VAR_INPUT
	m_Input_NumTextList:		INT;
END_VAR
    Rectangle (0,0 446x169), "%s", text list: 'TextList_Gaz', text index: m_Input_NumTextList
    Rectangle (361,0 85x25), "%s", text variable: m_Input_DG.CONF_Util_Name
    Frame (3,35 153x52)
        shows VISU_FCTS_SA(m_Input_ID_XML := 12, m_Input_UserRight := PRG_USER.ACTU_USER.FONCTION_SA AND NOT m_Input_Machine.STATE_Prod, m_Input_Operation := m_Input_Ligne.OP_MARCHE)
    Frame (3,106 153x52)
        shows VISU_FCTS_SA(m_Input_ID_XML := 13, m_Input_UserRight := PRG_USER.ACTU_USER.FONCTION_SA AND NOT m_Input_Machine.STATE_Prod, m_Input_Operation := m_Input_Ligne.OP_ARRET)
    Rectangle (170,99 91x24), "%s", text list: 'TextList_Gaz', text index: 3
    RoundedRectangle (354,99 87x24), "%1.1f", text variable: m_Input_DG.STATE_Flow
    RoundedRectangle (263,99 87x24), "%1.1f", text variable: m_Input_Ligne.PRM_Flow, input disabled if: (NOT PRG_USER.ACTU_USER.FONCTION_SA AND NOT m_Input_Machine.STATE_Prod) OR (NOT PRG_USER.ACTU_USER.MODIF_ENLIGNE AND m_Input_Machine.STATE_Prod)
        OnMouseClick: write the text variable via InputWithLimits, min 0, max m_Input_DG.CONF_Util_Max_Flow
    Rectangle (170,132 91x24), "%s", text list: 'TextList_Basiques', text index: 22
    RoundedRectangle (263,132 87x24), "%s", text variable: m_Input_Ligne.OP_RAMPE.PRM_Temps, input disabled if: (NOT PRG_USER.ACTU_USER.FONCTION_SA AND NOT m_Input_Machine.STATE_Prod) OR (NOT PRG_USER.ACTU_USER.MODIF_ENLIGNE AND m_Input_Machine.STATE_Prod)
        OnMouseClick: write the text variable via InputWithLimits
    Frame (163,35 153x52)
        shows VISU_FCTS_SA(m_Input_ID_XML := 14, m_Input_UserRight := PRG_USER.ACTU_USER.FONCTION_SA AND NOT m_Input_Machine.STATE_Prod, m_Input_Operation := m_Input_Ligne.OP_RAMPE.MARCHE)
    Button (323,35 120x50), "%s", input disabled if: (NOT PRG_USER.ACTU_USER.FONCTION_SA AND NOT m_Input_Machine.STATE_Prod) OR (NOT PRG_USER.ACTU_USER.MODIF_ENLIGNE AND m_Input_Machine.STATE_Prod), text list: 'TextList_Basiques', text index: 19
        toggle m_Input_Ligne.CO_Modif
    RoundedRectangle (354,132 87x24), "%s", text variable: m_Input_Ligne.OP_RAMPE.OUT_Tps_ecoule
END_VISUALIZATION

// ---- Visualizations/Semi Auto/Elements/SA_LIGNE_GAZ_MKS_RAMPE.TcVIS
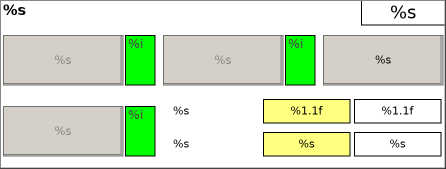
VISUALIZATION SA_LIGNE_GAZ_MKS_RAMPE  // 446x169
VAR_IN_OUT
	m_Input_Ligne:		BLOCK_LIGNE_GAZ;
	m_Input_Machine:	BLOCK_MODE_MARCHE_V2_0;
	m_Input_DG:			BLOCK_MFC_MKS_NoCoE;
	m_Input_UserRight:	BOOL;
END_VAR

VAR_INPUT
	m_Input_NumTextList:		INT;
END_VAR
    Rectangle (0,0 446x169), "%s", text list: 'TextList_Gaz', text index: m_Input_NumTextList
    Rectangle (361,0 85x25), "%s", text variable: m_Input_DG.CONF_Util_Name
    Frame (3,35 153x52)
        shows VISU_FCTS_SA(m_Input_ID_XML := 12, m_Input_UserRight := PRG_USER.ACTU_USER.FONCTION_SA AND NOT m_Input_Machine.STATE_Prod, m_Input_Operation := m_Input_Ligne.OP_MARCHE)
    Frame (3,106 153x52)
        shows VISU_FCTS_SA(m_Input_ID_XML := 13, m_Input_UserRight := PRG_USER.ACTU_USER.FONCTION_SA AND NOT m_Input_Machine.STATE_Prod, m_Input_Operation := m_Input_Ligne.OP_ARRET)
    Rectangle (170,99 91x24), "%s", text list: 'TextList_Gaz', text index: 3
    RoundedRectangle (354,99 87x24), "%1.1f", text variable: m_Input_DG.STATE_Flow
    RoundedRectangle (263,99 87x24), "%1.1f", text variable: m_Input_Ligne.PRM_Flow, input disabled if: (NOT PRG_USER.ACTU_USER.FONCTION_SA AND NOT m_Input_Machine.STATE_Prod) OR (NOT PRG_USER.ACTU_USER.MODIF_ENLIGNE AND m_Input_Machine.STATE_Prod)
        OnMouseClick: write the text variable via InputWithLimits, min 0, max m_Input_DG.CONF_Util_Max_Flow
    Rectangle (170,132 91x24), "%s", text list: 'TextList_Basiques', text index: 22
    RoundedRectangle (263,132 87x24), "%s", text variable: m_Input_Ligne.OP_RAMPE.PRM_Temps, input disabled if: (NOT PRG_USER.ACTU_USER.FONCTION_SA AND NOT m_Input_Machine.STATE_Prod) OR (NOT PRG_USER.ACTU_USER.MODIF_ENLIGNE AND m_Input_Machine.STATE_Prod)
        OnMouseClick: write the text variable via Edit
    Frame (163,35 153x52)
        shows VISU_FCTS_SA(m_Input_ID_XML := 14, m_Input_UserRight := PRG_USER.ACTU_USER.FONCTION_SA AND NOT m_Input_Machine.STATE_Prod, m_Input_Operation := m_Input_Ligne.OP_RAMPE.MARCHE)
    Button (323,35 120x50), "%s", input disabled if: (NOT PRG_USER.ACTU_USER.FONCTION_SA AND NOT m_Input_Machine.STATE_Prod) OR (NOT PRG_USER.ACTU_USER.MODIF_ENLIGNE AND m_Input_Machine.STATE_Prod), text list: 'TextList_Basiques', text index: 19
        toggle m_Input_Ligne.CO_Modif
    RoundedRectangle (354,132 87x24), "%s", text variable: m_Input_Ligne.OP_RAMPE.OUT_Tps_ecoule
END_VISUALIZATION

// ---- Visualizations/Semi Auto/Elements/SA_POMP_1E_PCR_PPM.TcVIS
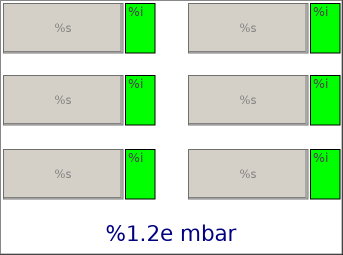
VISUALIZATION SA_POMP_1E_PCR_PPM  // 343x255
VAR_IN_OUT
	m_Input_PRG:		BLOCK_PRG_POMPAGE;
	m_Input_Jauge:		BLOCK_BCG450_ANA;
END_VAR
    Rectangle (0,0 343x255)
    Frame (3,75 153x52)
        shows VISU_FCTS_SA(m_Input_ID_XML := 0, m_Input_UserRight := PRG_USER.ACTU_USER.FONCTION_SA, m_Input_Operation := m_Input_PRG.POMPAGE.OP_Pompage_Sec)
    Frame (3,3 153x52)
        shows VISU_FCTS_SA(m_Input_ID_XML := 1, m_Input_UserRight := PRG_USER.ACTU_USER.FONCTION_SA, m_Input_Operation := m_Input_PRG.POMPAGE.OP_Marche_Pompes)
    Frame (188,3 153x52)
        shows VISU_FCTS_SA(m_Input_ID_XML := 2, m_Input_UserRight := PRG_USER.ACTU_USER.FONCTION_SA, m_Input_Operation := m_Input_PRG.POMPAGE.OP_Arret_Pompes)
    Frame (188,75 153x52)
        shows VISU_FCTS_SA(m_Input_ID_XML := 3, m_Input_UserRight := PRG_USER.ACTU_USER.FONCTION_SA, m_Input_Operation := m_Input_PRG.POMPAGE.OP_Isolement)
    Frame (3,149 153x52)
        shows VISU_FCTS_SA(m_Input_ID_XML := 4, m_Input_UserRight := PRG_USER.ACTU_USER.FONCTION_SA, m_Input_Operation := m_Input_PRG.POMPAGE.OP_Ventilation)
    Rectangle (80,219 182x29), "%1.2e mbar", text variable: m_Input_Jauge.STATE_Pression
    Frame (188,149 153x52)
        shows VISU_FCTS_SA(m_Input_ID_XML := 17, m_Input_UserRight := PRG_USER.ACTU_USER.FONCTION_SA, m_Input_Operation := m_Input_PRG.POMPAGE.OP_Regen)
END_VISUALIZATION

// ---- Visualizations/Semi Auto/Elements/SA_POMP_1E_PCR_PPM_ASS.TcVIS
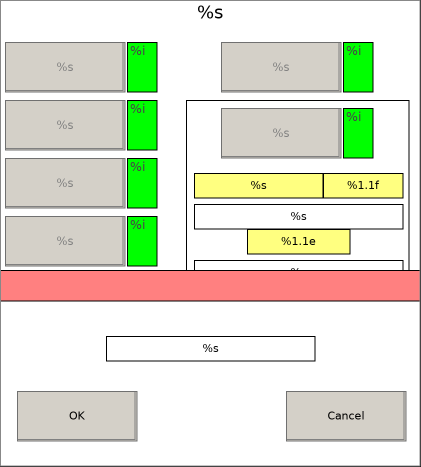
VISUALIZATION SA_POMP_1E_PCR_PPM_ASS  // 421x467
VAR_IN_OUT
	m_Input_PRG:			BLOCK_PRG_POMPAGE;
	m_Input_Jauge:			BLOCK_BCG450_ETHERCAT;
	m_Input_Process:		BLOCK_CDG_ETHERCAT;
	m_Input_Vanne:			BLOCK_VVAT_650_ETHERCAT;
	m_Input_Machine:		BLOCK_MODE_MARCHE_V2_0;
END_VAR
    Rectangle (0,0 421x467), "%s", text list: 'TextList_Navigation', text index: 6
    Frame (5,42 153x52)
        shows VISU_FCTS_SA(m_Input_ID_XML := 1, m_Input_UserRight := PRG_USER.ACTU_USER.FONCTION_SA, m_Input_Operation := m_Input_PRG.POMPAGE.OP_Marche_Pompes)
    Rectangle (74,391 63x25), "%s", text variable: m_Input_Jauge.MNEMO
    Rectangle (144,389 192x29), "%1.2e mbar", text variable: m_Input_Jauge.STATE_Pression
    Rectangle (74,425 63x25), "%s", text variable: m_Input_Process.MNEMO
    Rectangle (144,423 192x29), "%1.2e mbar", text variable: m_Input_Process.STATE_Pression
    Frame (5,100 153x52)
        shows VISU_FCTS_SA(m_Input_ID_XML := 0, m_Input_UserRight := PRG_USER.ACTU_USER.FONCTION_SA, m_Input_Operation := m_Input_PRG.POMPAGE.OP_Pompage_Sec)
    Frame (5,216 153x52)
        shows VISU_FCTS_SA(m_Input_ID_XML := 3, m_Input_UserRight := PRG_USER.ACTU_USER.FONCTION_SA, m_Input_Operation := m_Input_PRG.POMPAGE.OP_Isolement)
    Frame (4,334 153x52)
        shows VISU_FCTS_SA(m_Input_ID_XML := 17, m_Input_UserRight := FALSE, m_Input_Operation := m_Input_PRG.POMPAGE.OP_Regen)
    Frame (5,274 153x52)
        shows VISU_FCTS_SA(m_Input_ID_XML := 4, m_Input_UserRight := PRG_USER.ACTU_USER.FONCTION_SA, m_Input_Operation := m_Input_PRG.POMPAGE.OP_Ventilation)
    Rectangle (186,100 223x274)
    Frame (221,108 153x52)
        shows VISU_FCTS_SA(m_Input_ID_XML := 11, m_Input_UserRight := PRG_USER.ACTU_USER.FONCTION_SA, m_Input_Operation := m_Input_PRG.POMPAGE.OP_Pompage_Proc)
    RoundedRectangle (194,173 129x25), "%s", invisible if: NOT m_Input_Vanne.PRM_Mode, input disabled if: NOT (PRG_USER.ACTU_USER.FONCTION_SA AND NOT m_Input_MACHINE.STATE_Prod) OR m_Input_MACHINE.STATE_Prod, text list: 'TextList_VVAT_650_ETHERCAT', text index: 8
        OnMouseClick: toggle m_Input_Vanne.PRM_Mode
    RoundedRectangle (194,173 129x25), "%s", invisible if: m_Input_Vanne.PRM_Mode, input disabled if: NOT (PRG_USER.ACTU_USER.FONCTION_SA AND NOT m_Input_MACHINE.STATE_Prod) OR m_Input_MACHINE.STATE_Prod, text list: 'TextList_VVAT_650_ETHERCAT', text index: 7
        OnMouseClick: toggle m_Input_Vanne.PRM_Mode
    RoundedRectangle (194,204 209x25), "%s", invisible if: NOT m_Input_Vanne.PRM_Mode, text list: 'TextList_VVAT_650_ETHERCAT', text index: 4
    RoundedRectangle (194,260 209x25), "%s", invisible if: NOT m_Input_Vanne.PRM_Mode, text list: 'TextList_VVAT_650_ETHERCAT', text index: 5
    RoundedRectangle (194,316 209x25), "%s", invisible if: NOT m_Input_Vanne.PRM_Mode, text list: 'TextList_VVAT_650_ETHERCAT', text index: 6
    RoundedRectangle (247,341 103x25), "%s", text variable: m_Input_Vanne.PRM_Tim_W_Pr, invisible if: NOT m_Input_Vanne.PRM_Mode, input disabled if: NOT (PRG_USER.ACTU_USER.FONCTION_SA AND NOT m_Input_MACHINE.STATE_Prod) OR m_Input_MACHINE.STATE_Prod
        OnMouseClick: write the text variable via InputWithLimits
    RoundedRectangle (247,285 103x25), "%1.1e", text variable: m_Input_Vanne.PRM_W_Pr_HI, invisible if: NOT m_Input_Vanne.PRM_Mode, input disabled if: NOT (PRG_USER.ACTU_USER.FONCTION_SA AND NOT m_Input_MACHINE.STATE_Prod) OR m_Input_MACHINE.STATE_Prod
        OnMouseClick: write the text variable via InputWithLimits, min 0, max 1000
    RoundedRectangle (247,229 103x25), "%1.1e", text variable: m_Input_Vanne.PRM_W_Pr_LO, invisible if: NOT m_Input_Vanne.PRM_Mode, input disabled if: NOT (PRG_USER.ACTU_USER.FONCTION_SA AND NOT m_Input_MACHINE.STATE_Prod) OR m_Input_MACHINE.STATE_Prod
        OnMouseClick: write the text variable via InputWithLimits, min 0, max 1000
    RoundedRectangle (323,173 80x25), "%1.1e", text variable: m_Input_Vanne.PRM_Pression, invisible if: NOT m_Input_Vanne.PRM_Mode, input disabled if: NOT (PRG_USER.ACTU_USER.FONCTION_SA AND NOT m_Input_MACHINE.STATE_Prod) OR m_Input_MACHINE.STATE_Prod
        OnMouseClick: write the text variable via InputWithLimits, min 0, max 1000
    RoundedRectangle (323,173 80x25), "%1.1f", text variable: m_Input_Vanne.PRM_Position, invisible if: m_Input_Vanne.PRM_Mode, input disabled if: NOT (PRG_USER.ACTU_USER.FONCTION_SA AND NOT m_Input_MACHINE.STATE_Prod) OR m_Input_MACHINE.STATE_Prod
        OnMouseClick: write the text variable via InputWithLimits, min 0, max 100
    Frame (221,42 153x52)
        shows VISU_FCTS_SA(m_Input_ID_XML := 2, m_Input_UserRight := PRG_USER.ACTU_USER.FONCTION_SA, m_Input_Operation := m_Input_PRG.POMPAGE.OP_Arret_Pompes)
    Frame (5,158 153x52)
        shows VISU_FCTS_SA(m_Input_ID_XML := 28, m_Input_UserRight := PRG_USER.ACTU_USER.FONCTION_SA, m_Input_Operation := m_Input_PRG.POMPAGE.OP_Pompage_Prim)
    Button (4,334 120x50), "%s", input disabled if: NOT m_Input_PRG.POMPAGE.OP_Regen.Autor_IHM OR NOT (PRG_USER.ACTU_USER.FONCTION_SA AND NOT m_Input_Machine.STATE_PROD), text list: 'TextList_SA_Operations', text index: 17
        OnMouseClick: execute { Global_Variables.SHOW_CONFIRM_REGEN:=(TRUE); }
    Group (0,270 421x197), invisible if: NOT Global_Variables.SHOW_CONFIRM_REGEN
        Rectangle (0,0 421x197)
        Button (17,121 120x50), "OK", input disabled if: NOT m_Input_PRG.POMPAGE.OP_Regen.Autor_IHM OR NOT (PRG_USER.ACTU_USER.FONCTION_SA AND NOT m_Input_Machine.STATE_PROD)
            OnMouseClick: execute { m_Input_PRG.POMPAGE.OP_Regen.ON_IHM:=(TRUE); Global_Variables.SHOW_CONFIRM_REGEN:=(FALSE); }
        Button (286,121 120x50), "Cancel"
            OnMouseClick: execute { Global_Variables.SHOW_CONFIRM_REGEN:=(FALSE); }
        Rectangle (0,0 421x31)
        RoundedRectangle (106,66 209x25), "%s", text list: 'TextList_Pompage', text index: 1
END_VISUALIZATION

// ---- Visualizations/Semi Auto/Elements/SA_POMP_1E_PCR_PPM_ASS_M11.TcVIS
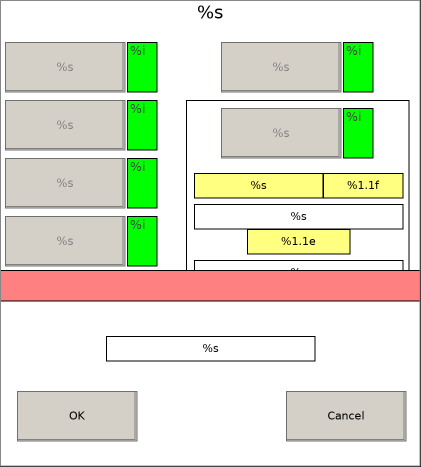
VISUALIZATION SA_POMP_1E_PCR_PPM_ASS_M11  // 421x467
VAR_IN_OUT
	m_Input_PRG:			BLOCK_PRG_POMPAGE;
	m_Input_Jauge:			BLOCK_BCG450_ETHERCAT;
	m_Input_Vanne:			BLOCK_VVAT_650_NO;
	m_Input_Machine:		BLOCK_MODE_MARCHE_V2_0;
END_VAR
    Rectangle (0,0 421x467), "%s", text list: 'TextList_Navigation', text index: 6
    Frame (5,42 153x52)
        shows VISU_FCTS_SA(m_Input_ID_XML := 1, m_Input_UserRight := PRG_USER.ACTU_USER.FONCTION_SA, m_Input_Operation := m_Input_PRG.POMPAGE.OP_Marche_Pompes)
    Rectangle (74,391 63x25), "%s", text variable: m_Input_Jauge.MNEMO
    Rectangle (144,389 192x29), "%1.2e mbar", text variable: m_Input_Jauge.STATE_Pression
    Frame (5,100 153x52)
        shows VISU_FCTS_SA(m_Input_ID_XML := 0, m_Input_UserRight := PRG_USER.ACTU_USER.FONCTION_SA, m_Input_Operation := m_Input_PRG.POMPAGE.OP_Pompage_Sec)
    Frame (5,216 153x52)
        shows VISU_FCTS_SA(m_Input_ID_XML := 3, m_Input_UserRight := PRG_USER.ACTU_USER.FONCTION_SA, m_Input_Operation := m_Input_PRG.POMPAGE.OP_Isolement)
    Frame (4,334 153x52)
        shows VISU_FCTS_SA(m_Input_ID_XML := 17, m_Input_UserRight := FALSE, m_Input_Operation := m_Input_PRG.POMPAGE.OP_Regen)
    Frame (5,274 153x52)
        shows VISU_FCTS_SA(m_Input_ID_XML := 4, m_Input_UserRight := PRG_USER.ACTU_USER.FONCTION_SA, m_Input_Operation := m_Input_PRG.POMPAGE.OP_Ventilation)
    Rectangle (186,100 223x274)
    Frame (221,108 153x52)
        shows VISU_FCTS_SA(m_Input_ID_XML := 11, m_Input_UserRight := PRG_USER.ACTU_USER.FONCTION_SA, m_Input_Operation := m_Input_PRG.POMPAGE.OP_Pompage_Proc)
    RoundedRectangle (194,173 129x25), "%s", invisible if: NOT m_Input_Vanne.PRM_Mode, input disabled if: NOT (PRG_USER.ACTU_USER.FONCTION_SA AND NOT m_Input_MACHINE.STATE_Prod) OR m_Input_MACHINE.STATE_Prod, text list: 'TextList_VVAT_650_ETHERCAT', text index: 8
        OnMouseClick: toggle m_Input_Vanne.PRM_Mode
    RoundedRectangle (194,173 129x25), "%s", invisible if: m_Input_Vanne.PRM_Mode, input disabled if: NOT (PRG_USER.ACTU_USER.FONCTION_SA AND NOT m_Input_MACHINE.STATE_Prod) OR m_Input_MACHINE.STATE_Prod, text list: 'TextList_VVAT_650_ETHERCAT', text index: 7
        OnMouseClick: toggle m_Input_Vanne.PRM_Mode
    RoundedRectangle (194,204 209x25), "%s", invisible if: NOT m_Input_Vanne.PRM_Mode, text list: 'TextList_VVAT_650_ETHERCAT', text index: 4
    RoundedRectangle (194,260 209x25), "%s", invisible if: NOT m_Input_Vanne.PRM_Mode, text list: 'TextList_VVAT_650_ETHERCAT', text index: 5
    RoundedRectangle (194,316 209x25), "%s", invisible if: NOT m_Input_Vanne.PRM_Mode, text list: 'TextList_VVAT_650_ETHERCAT', text index: 6
    RoundedRectangle (247,341 103x25), "%s", text variable: m_Input_Vanne.PRM_Tim_W_Pr, invisible if: NOT m_Input_Vanne.PRM_Mode, input disabled if: NOT (PRG_USER.ACTU_USER.FONCTION_SA AND NOT m_Input_MACHINE.STATE_Prod) OR m_Input_MACHINE.STATE_Prod
        OnMouseClick: write the text variable via InputWithLimits
    RoundedRectangle (247,285 103x25), "%1.1e", text variable: m_Input_Vanne.PRM_W_Pr_HI, invisible if: NOT m_Input_Vanne.PRM_Mode, input disabled if: NOT (PRG_USER.ACTU_USER.FONCTION_SA AND NOT m_Input_MACHINE.STATE_Prod) OR m_Input_MACHINE.STATE_Prod
        OnMouseClick: write the text variable via InputWithLimits, min 0, max 1000
    RoundedRectangle (247,229 103x25), "%1.1e", text variable: m_Input_Vanne.PRM_W_Pr_LO, invisible if: NOT m_Input_Vanne.PRM_Mode, input disabled if: NOT (PRG_USER.ACTU_USER.FONCTION_SA AND NOT m_Input_MACHINE.STATE_Prod) OR m_Input_MACHINE.STATE_Prod
        OnMouseClick: write the text variable via InputWithLimits, min 0, max 1000
    RoundedRectangle (323,173 80x25), "%1.1e", text variable: m_Input_Vanne.PRM_Pression, invisible if: NOT m_Input_Vanne.PRM_Mode, input disabled if: NOT (PRG_USER.ACTU_USER.FONCTION_SA AND NOT m_Input_MACHINE.STATE_Prod) OR m_Input_MACHINE.STATE_Prod
        OnMouseClick: write the text variable via InputWithLimits, min 0, max 1000
    RoundedRectangle (323,173 80x25), "%1.1f", text variable: m_Input_Vanne.PRM_Position, invisible if: m_Input_Vanne.PRM_Mode, input disabled if: NOT (PRG_USER.ACTU_USER.FONCTION_SA AND NOT m_Input_MACHINE.STATE_Prod) OR m_Input_MACHINE.STATE_Prod
        OnMouseClick: write the text variable via InputWithLimits, min 0, max 100
    Frame (221,42 153x52)
        shows VISU_FCTS_SA(m_Input_ID_XML := 2, m_Input_UserRight := PRG_USER.ACTU_USER.FONCTION_SA, m_Input_Operation := m_Input_PRG.POMPAGE.OP_Arret_Pompes)
    Frame (5,158 153x52)
        shows VISU_FCTS_SA(m_Input_ID_XML := 28, m_Input_UserRight := PRG_USER.ACTU_USER.FONCTION_SA, m_Input_Operation := m_Input_PRG.POMPAGE.OP_Pompage_Prim)
    Button (4,334 120x50), "%s", input disabled if: NOT m_Input_PRG.POMPAGE.OP_Regen.Autor_IHM OR NOT (PRG_USER.ACTU_USER.FONCTION_SA AND NOT m_Input_Machine.STATE_PROD), text list: 'TextList_SA_Operations', text index: 17
        OnMouseClick: execute { Global_Variables.SHOW_CONFIRM_REGEN:=(TRUE); }
    Group (0,270 421x197), invisible if: NOT Global_Variables.SHOW_CONFIRM_REGEN
        Rectangle (0,0 421x197)
        Button (17,121 120x50), "OK", input disabled if: NOT m_Input_PRG.POMPAGE.OP_Regen.Autor_IHM OR NOT (PRG_USER.ACTU_USER.FONCTION_SA AND NOT m_Input_Machine.STATE_PROD)
            OnMouseClick: execute { m_Input_PRG.POMPAGE.OP_Regen.ON_IHM:=(TRUE); Global_Variables.SHOW_CONFIRM_REGEN:=(FALSE); }
        Button (286,121 120x50), "Cancel"
            OnMouseClick: execute { Global_Variables.SHOW_CONFIRM_REGEN:=(FALSE); }
        Rectangle (0,0 421x31)
        RoundedRectangle (106,66 209x25), "%s", text list: 'TextList_Pompage', text index: 1
END_VISUALIZATION

// ---- Visualizations/Semi Auto/Elements/SA_POMP_2E_PCR_PPM_ASS.TcVIS
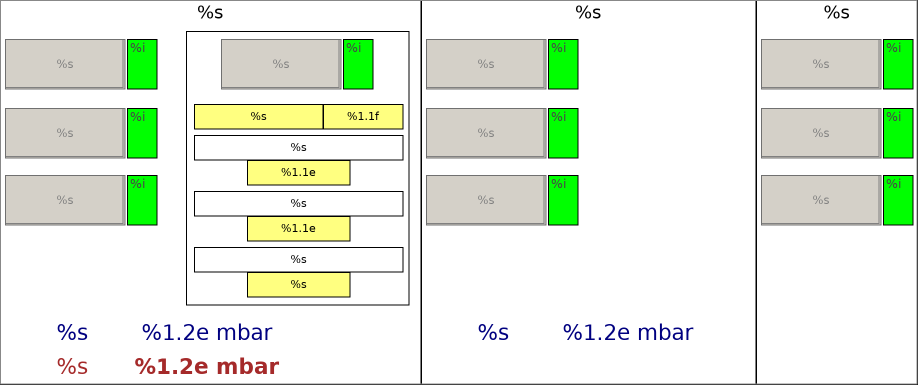
VISUALIZATION SA_POMP_2E_PCR_PPM_ASS  // 918x385
VAR_IN_OUT
	m_Input_PRG:			BLOCK_PRG_POMPAGE;
	m_Input_Jauge:			BLOCK_BCG450_ETHERCAT;
	m_Input_Process:		BLOCK_CDG_ETHERCAT;
	m_Input_Pr_Sas:			BLOCK_PCG550_ETHERCAT;
	m_Input_Vanne:			BLOCK_VVAT_650_ETHERCAT;
	m_Input_Machine:		BLOCK_MODE_MARCHE;
END_VAR
    Rectangle (0,0 421x385), "%s", text list: 'TextList_Navigation', text index: 6
    Rectangle (421,0 335x385), "%s", text list: 'TextList_Navigation', text index: 7
    Rectangle (756,0 162x385), "%s", text list: 'TextList_Navigation', text index: 13
    Frame (761,39 153x52)
        shows VISU_FCTS_SA(m_Input_ID_XML := 1, m_Input_UserRight := PRG_USER.ACTU_USER.FONCTION_SA, m_Input_Operation := m_Input_PRG.POMPAGE.OP_Marche_Pompes)
    Frame (761,108 153x52)
        shows VISU_FCTS_SA(m_Input_ID_XML := 2, m_Input_UserRight := PRG_USER.ACTU_USER.FONCTION_SA, m_Input_Operation := m_Input_PRG.POMPAGE.OP_Arret_Pompes)
    Rectangle (41,320 63x25), "%s", text variable: m_Input_Jauge.MNEMO
    Rectangle (111,318 192x29), "%1.2e mbar", text variable: m_Input_Jauge.STATE_Pression
    Rectangle (41,354 63x25), "%s", text variable: m_Input_Process.MNEMO
    Rectangle (111,352 192x29), "%1.2e mbar", text variable: m_Input_Process.STATE_Pression
    Frame (5,39 153x52)
        shows VISU_FCTS_SA(m_Input_ID_XML := 0, m_Input_UserRight := PRG_USER.ACTU_USER.FONCTION_SA, m_Input_Operation := m_Input_PRG.POMPAGE.OP_Pompage_Sec)
    Frame (426,39 153x52)
        shows VISU_FCTS_SA(m_Input_ID_XML := 0, m_Input_UserRight := PRG_USER.ACTU_USER.PRODUCTION, m_Input_Operation := m_Input_PRG.POMPAGE.OP_Pompage_SAS)
    Frame (5,108 153x52)
        shows VISU_FCTS_SA(m_Input_ID_XML := 3, m_Input_UserRight := PRG_USER.ACTU_USER.FONCTION_SA, m_Input_Operation := m_Input_PRG.POMPAGE.OP_Isolement)
    Frame (426,108 153x52)
        shows VISU_FCTS_SA(m_Input_ID_XML := 3, m_Input_UserRight := PRG_USER.ACTU_USER.FONCTION_SA, m_Input_Operation := m_Input_PRG.POMPAGE.OP_Isolement_SAS)
    Frame (761,175 153x52)
        shows VISU_FCTS_SA(m_Input_ID_XML := 17, m_Input_UserRight := PRG_USER.ACTU_USER.FONCTION_SA, m_Input_Operation := m_Input_PRG.POMPAGE.OP_Regen)
    Frame (5,175 153x52)
        shows VISU_FCTS_SA(m_Input_ID_XML := 4, m_Input_UserRight := PRG_USER.ACTU_USER.FONCTION_SA, m_Input_Operation := m_Input_PRG.POMPAGE.OP_Ventilation)
    Frame (426,175 153x52)
        shows VISU_FCTS_SA(m_Input_ID_XML := 4, m_Input_UserRight := PRG_USER.ACTU_USER.PRODUCTION, m_Input_Operation := m_Input_PRG.POMPAGE.OP_Ventilation_SAS)
    Rectangle (462,320 63x25), "%s", text variable: m_Input_Pr_Sas.MNEMO
    Rectangle (532,318 192x29), "%1.2e mbar", text variable: m_Input_Pr_Sas.STATE_Pression
    Rectangle (186,31 223x274)
    Frame (221,39 153x52)
        shows VISU_FCTS_SA(m_Input_ID_XML := 11, m_Input_UserRight := PRG_USER.ACTU_USER.FONCTION_SA, m_Input_Operation := m_Input_PRG.POMPAGE.OP_Pompage_Proc)
    RoundedRectangle (194,104 129x25), "%s", invisible if: NOT m_Input_Vanne.PRM_Mode, input disabled if: NOT (PRG_USER.ACTU_USER.FONCTION_SA AND NOT m_Input_MACHINE.STATE_Prod) OR m_Input_MACHINE.STATE_Prod, text list: 'TextList_VVAT_650_ETHERCAT', text index: 8
        OnMouseClick: toggle m_Input_Vanne.PRM_Mode
    RoundedRectangle (194,104 129x25), "%s", invisible if: m_Input_Vanne.PRM_Mode, input disabled if: NOT (PRG_USER.ACTU_USER.FONCTION_SA AND NOT m_Input_MACHINE.STATE_Prod) OR m_Input_MACHINE.STATE_Prod, text list: 'TextList_VVAT_650_ETHERCAT', text index: 7
        OnMouseClick: toggle m_Input_Vanne.PRM_Mode
    RoundedRectangle (194,135 209x25), "%s", invisible if: NOT m_Input_Vanne.PRM_Mode, text list: 'TextList_VVAT_650_ETHERCAT', text index: 4
    RoundedRectangle (194,191 209x25), "%s", invisible if: NOT m_Input_Vanne.PRM_Mode, text list: 'TextList_VVAT_650_ETHERCAT', text index: 5
    RoundedRectangle (194,247 209x25), "%s", invisible if: NOT m_Input_Vanne.PRM_Mode, text list: 'TextList_VVAT_650_ETHERCAT', text index: 6
    RoundedRectangle (247,272 103x25), "%s", text variable: m_Input_Vanne.PRM_Tim_W_Pr, invisible if: NOT m_Input_Vanne.PRM_Mode, input disabled if: NOT (PRG_USER.ACTU_USER.FONCTION_SA AND NOT m_Input_MACHINE.STATE_Prod) OR m_Input_MACHINE.STATE_Prod
        OnMouseClick: write the text variable via VisuDialogs.Keypad
    RoundedRectangle (247,216 103x25), "%1.1e", text variable: m_Input_Vanne.PRM_W_Pr_HI, invisible if: NOT m_Input_Vanne.PRM_Mode, input disabled if: NOT (PRG_USER.ACTU_USER.FONCTION_SA AND NOT m_Input_MACHINE.STATE_Prod) OR m_Input_MACHINE.STATE_Prod
        OnMouseClick: write the text variable via VisuDialogs.Numpad, min 0, max 1000
    RoundedRectangle (247,160 103x25), "%1.1e", text variable: m_Input_Vanne.PRM_W_Pr_LO, invisible if: NOT m_Input_Vanne.PRM_Mode, input disabled if: NOT (PRG_USER.ACTU_USER.FONCTION_SA AND NOT m_Input_MACHINE.STATE_Prod) OR m_Input_MACHINE.STATE_Prod
        OnMouseClick: write the text variable via VisuDialogs.Numpad, min 0, max 1000
    RoundedRectangle (323,104 80x25), "%1.1e", text variable: m_Input_Vanne.PRM_Pression, invisible if: NOT m_Input_Vanne.PRM_Mode, input disabled if: NOT (PRG_USER.ACTU_USER.FONCTION_SA AND NOT m_Input_MACHINE.STATE_Prod) OR m_Input_MACHINE.STATE_Prod
        OnMouseClick: write the text variable via VisuDialogs.Numpad, min 0, max 1000
    RoundedRectangle (323,104 80x25), "%1.1f", text variable: m_Input_Vanne.PRM_Position, invisible if: m_Input_Vanne.PRM_Mode, input disabled if: NOT (PRG_USER.ACTU_USER.FONCTION_SA AND NOT m_Input_MACHINE.STATE_Prod) OR m_Input_MACHINE.STATE_Prod
        OnMouseClick: write the text variable via VisuDialogs.Numpad, min 0, max 100
END_VISUALIZATION

// ---- Visualizations/Semi Auto/Elements/SA_POMP_ENCEINTE.TcVIS
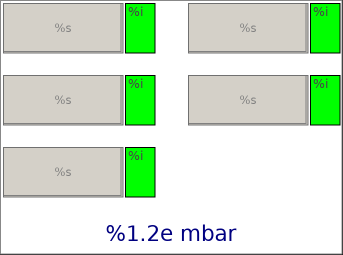
VISUALIZATION SA_POMP_ENCEINTE  // 343x255
VAR_IN_OUT
	m_Input_PRG:		BLOCK_PRG_POMPAGE;
	m_Input_Jauge:		BLOCK_BCG450_ETHERCAT;
END_VAR
    Rectangle (0,0 343x255)
    Frame (3,75 153x52)
        shows VISU_FCTS_SA(m_Input_ID_XML := 0, m_Input_UserRight := PRG_USER.ACTU_USER.FONCTION_SA, m_Input_Operation := m_Input_PRG.POMPAGE.OP_Pompage_Sec)
    Frame (3,3 153x52)
        shows VISU_FCTS_SA(m_Input_ID_XML := 1, m_Input_UserRight := PRG_USER.ACTU_USER.FONCTION_SA, m_Input_Operation := m_Input_PRG.POMPAGE.OP_Marche_Pompes)
    Frame (188,3 153x52)
        shows VISU_FCTS_SA(m_Input_ID_XML := 2, m_Input_UserRight := PRG_USER.ACTU_USER.FONCTION_SA, m_Input_Operation := m_Input_PRG.POMPAGE.OP_Arret_Pompes)
    Frame (188,75 153x52)
        shows VISU_FCTS_SA(m_Input_ID_XML := 3, m_Input_UserRight := PRG_USER.ACTU_USER.FONCTION_SA, m_Input_Operation := m_Input_PRG.POMPAGE.OP_Isolement)
    Frame (3,147 153x52)
        shows VISU_FCTS_SA(m_Input_ID_XML := 4, m_Input_UserRight := PRG_USER.ACTU_USER.FONCTION_SA, m_Input_Operation := m_Input_PRG.POMPAGE.OP_Ventilation)
    Rectangle (80,219 182x29), "%1.2e mbar", text variable: m_Input_Jauge.STATE_Pression
END_VISUALIZATION

// ---- Visualizations/Semi Auto/Elements/SA_POMP_SAS.TcVIS
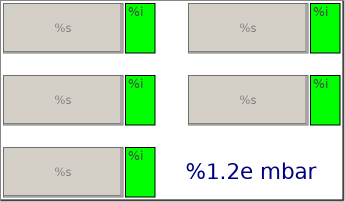
VISUALIZATION SA_POMP_SAS  // 345x202
VAR_IN_OUT
	m_Input_PRG:		BLOCK_PRG_POMPAGE_SAS;
	m_Input_Jauge:		BLOCK_BCG450_ETHERCAT;
END_VAR
    Rectangle (0,0 343x200)
    Frame (3,75 153x52)
        shows VISU_FCTS_SA(m_Input_ID_XML := 0, m_Input_UserRight := PRG_USER.ACTU_USER.FONCTION_SA, m_Input_Operation := m_Input_PRG.POMPAGE.OP_Pompage_Sec)
    Frame (3,3 153x52)
        shows VISU_FCTS_SA(m_Input_ID_XML := 1, m_Input_UserRight := PRG_USER.ACTU_USER.FONCTION_SA, m_Input_Operation := m_Input_PRG.POMPAGE.OP_Marche_Pompes)
    Frame (188,3 153x52)
        shows VISU_FCTS_SA(m_Input_ID_XML := 2, m_Input_UserRight := PRG_USER.ACTU_USER.FONCTION_SA, m_Input_Operation := m_Input_PRG.POMPAGE.OP_Arret_Pompes)
    Frame (188,75 153x52)
        shows VISU_FCTS_SA(m_Input_ID_XML := 3, m_Input_UserRight := PRG_USER.ACTU_USER.FONCTION_SA, m_Input_Operation := m_Input_PRG.POMPAGE.OP_Isolement)
    Frame (3,147 153x52)
        shows VISU_FCTS_SA(m_Input_ID_XML := 4, m_Input_UserRight := PRG_USER.ACTU_USER.FONCTION_SA, m_Input_Operation := m_Input_PRG.POMPAGE.OP_Ventilation)
    Rectangle (160,157 182x29), "%1.2e mbar", text variable: m_Input_Jauge.STATE_Pression
END_VISUALIZATION

// ---- Visualizations/Semi Auto/Elements/SA_PS.TcVIS
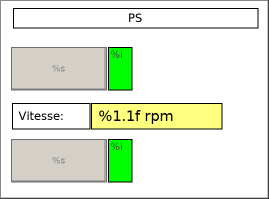
VISUALIZATION SA_PS  // 269x199
    Rectangle (0,0 269x199)
    Rectangle (12,103 78x26), "Vitesse:"
    Rectangle (13,8 245x20), "PS"
    Rectangle (91,103 131x26), "%1.1f rpm", text variable: PRG_MOUVEMENT_PS.ROTATION_PS.PRM_Vitesse, input disabled if: ((NOT PRG_User.ACTU_USER.MAINTENANCE AND NOT PRG_User.ACTU_USER.FONCTION_SA AND NOT PRG_User.ACTU_USER.MODIF_ENLIGNE) OR (NOT MACHINE.STATE_Wait_Prod AND NOT MACHINE.STATE_Manu)) <> 0
        OnMouseDown: write the text variable via InputWithLimits, min 0.2, max 20.0
    Frame (11,47 123x45)
        shows VISU_FCTS_SA(m_Input_ID_XML := 15, m_Input_UserRight := PRG_USER.ACTU_USER.FONCTION_SA, m_Input_Operation := PRG_MOUVEMENT_PS.ROTATION_PS.OP_Rotation)
    Frame (11,139 123x45)
        shows VISU_FCTS_SA(m_Input_ID_XML := 7, m_Input_UserRight := PRG_USER.ACTU_USER.FONCTION_SA, m_Input_Operation := PRG_MOUVEMENT_PS.ROTATION_PS.OP_Stop)
END_VISUALIZATION

// ---- Visualizations/Semi Auto/Elements/SA_REGUL_GAZ.TcVIS
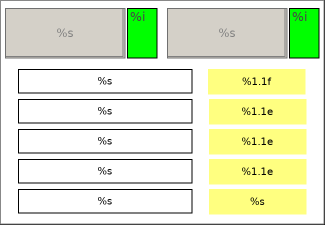
VISUALIZATION SA_REGUL_GAZ  // 325x225
VAR_IN_OUT
	m_Input_REGULATION : BLOCK_REGUL_PR_GAZ;
	m_Input_MACHINE : BLOCK_MODE_MARCHE_V2_0;
END_VAR
    Rectangle (0,0 325x225)
    Frame (5,8 158x57)
        shows VISU_FCTS_SA(m_Input_ID_XML := 29, m_Input_Operation := m_Input_REGULATION.OP_MARCHE, m_Input_UserRight := Global_Variables.PRG_USER.ACTU_USER.FONCTION_SA AND NOT m_Input_MACHINE.STATE_PROD)
    RoundedRectangle (18,69 174x24), "%s", text list: 'TextList_Gaz', text index: 15
    RoundedRectangle (208,69 97x25), "%1.1f", text variable: m_Input_REGULATION.PRM_Pos_Vanne, input disabled if: ((NOT PRG_User.ACTU_USER.FONCTION_SA AND NOT m_Input_MACHINE.STATE_PROD) OR (NOT PRG_User.ACTU_USER.MODIF_ENLIGNE AND m_Input_MACHINE.STATE_PROD)) <> 0
        OnMouseDown: write the text variable via InputWithLimits, min 0, max 100
    Frame (167,8 157x56)
        shows VISU_FCTS_SA(m_Input_ID_XML := 7, m_Input_Operation := m_Input_REGULATION.OP_ARRET, m_Input_UserRight := Global_Variables.PRG_USER.ACTU_USER.FONCTION_SA AND NOT m_Input_MACHINE.STATE_PROD)
    RoundedRectangle (18,99 174x24), "%s", text list: 'TextList_Gaz', text index: 16
    RoundedRectangle (209,99 97x25), "%1.1e", text variable: m_Input_REGULATION.PRM_Pressure, input disabled if: ((NOT PRG_User.ACTU_USER.FONCTION_SA AND NOT m_Input_MACHINE.STATE_PROD) OR (NOT PRG_User.ACTU_USER.MODIF_ENLIGNE AND m_Input_MACHINE.STATE_PROD)) <> 0
        OnMouseDown: write the text variable via InputWithLimits, min 0, max 1000
    RoundedRectangle (18,129 174x24), "%s", text list: 'TextList_Gaz', text index: 17
    RoundedRectangle (209,129 97x25), "%1.1e", text variable: m_Input_REGULATION.PRM_Pressure_L, input disabled if: ((NOT PRG_User.ACTU_USER.FONCTION_SA AND NOT m_Input_MACHINE.STATE_PROD) OR (NOT PRG_User.ACTU_USER.MODIF_ENLIGNE AND m_Input_MACHINE.STATE_PROD)) <> 0
        OnMouseDown: write the text variable via InputWithLimits, min 0, max 1000
    RoundedRectangle (18,159 174x24), "%s", text list: 'TextList_Gaz', text index: 18
    RoundedRectangle (209,159 97x25), "%1.1e", text variable: m_Input_REGULATION.PRM_Pressure_H, input disabled if: ((NOT PRG_User.ACTU_USER.FONCTION_SA AND NOT m_Input_MACHINE.STATE_PROD) OR (NOT PRG_User.ACTU_USER.MODIF_ENLIGNE AND m_Input_MACHINE.STATE_PROD)) <> 0
        OnMouseDown: write the text variable via InputWithLimits, min 0, max 1000
    RoundedRectangle (18,189 174x24), "%s", text list: 'TextList_Gaz', text index: 19
    RoundedRectangle (209,189 97x25), "%s", text variable: m_Input_REGULATION.PRM_Tim_Stab, input disabled if: ((NOT PRG_User.ACTU_USER.FONCTION_SA AND NOT m_Input_MACHINE.STATE_PROD) OR (NOT PRG_User.ACTU_USER.MODIF_ENLIGNE AND m_Input_MACHINE.STATE_PROD)) <> 0
        OnMouseDown: write the text variable via InputWithLimits
END_VISUALIZATION

// ---- Visualizations/Semi Auto/Elements/SA_ROT.TcVIS
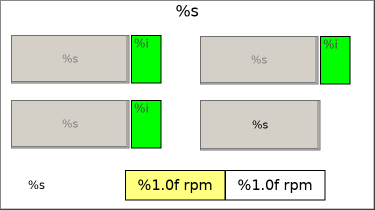
VISUALIZATION SA_ROT  // 375x210
VAR_IN_OUT
	m_Input_ROT:				BLOCK_ROTATION_CONTINUE_ATV;
	m_Input_PRG:				BLOCK_PRG_MOUVEMENT_PS;
END_VAR
    Rectangle (0,0 375x210), "%s", text list: 'TextList_Type_Moteur', text index: 1
    Button (200,100 120x50), "%s", input disabled if: not PRG_USER.ACTU_USER.FONCTION_SA, text list: 'TextList_Basiques', text index: 19
        tap m_Input_ROT.CO_Modif
    RoundedRectangle (125,170 100x30), "%1.0f rpm", text variable: m_Input_ROT.PRM_vitesse, input disabled if: (NOT PRG_User.ACTU_USER.MAINTENANCE AND NOT PRG_User.ACTU_USER.FONCTION_SA AND NOT PRG_User.ACTU_USER.MODIF_ENLIGNE) OR ( MACHINE.STATE_Manu )
        OnMouseDown: write the text variable via InputWithLimits, min m_Input_ROT.CONF_VMIN, max m_Input_ROT.CONF_VMAX, title 'Speed'
    Rectangle (25,170 100x30), "%s", text list: 'TextList_Moteurs', text index: 7
    RoundedRectangle (225,170 100x30), "%1.0f rpm", text variable: m_Input_ROT.STATE_Vitesse
    Frame (11,35 152x50), invisible if: not m_Input_PRG.CONF_Rotation
        shows VISU_FCTS_SA(m_Input_ID_XML := 15, m_Input_Operation := m_Input_ROT.OP_ROTATION, m_Input_UserRight := PRG_USER.ACTU_USER.FONCTION_SA AND NOT MACHINE.STATE_Prod)
        p768090162: m_Input_ROT.OP_ROTATION
        p1726406813: PRG_USER.ACTU_USER.FONCTION_SA AND NOT MACHINE.STATE_Prod
    Frame (200,36 152x50)
        shows VISU_FCTS_SA(m_Input_ID_XML := 7, m_Input_Operation := m_Input_ROT.OP_ARRET, m_Input_UserRight := PRG_USER.ACTU_USER.FONCTION_SA AND NOT MACHINE.STATE_Prod)
        p768090162: m_Input_ROT.OP_ARRET
        p1726406813: PRG_USER.ACTU_USER.FONCTION_SA AND NOT MACHINE.STATE_Prod
    Frame (11,100 152x50), invisible if: not m_Input_PRG.CONF_Positionnement
        shows VISU_FCTS_SA(m_Input_ID_XML := 8, m_Input_Operation := m_Input_ROT.OP_POSITION, m_Input_UserRight := PRG_USER.ACTU_USER.FONCTION_SA AND NOT MACHINE.STATE_Prod)
        p768090162: m_Input_ROT.OP_POSITION
        p1726406813: PRG_USER.ACTU_USER.FONCTION_SA AND NOT MACHINE.STATE_Prod
END_VISUALIZATION

// ---- Visualizations/Semi Auto/Elements/SA_TEST_RP.TcVIS
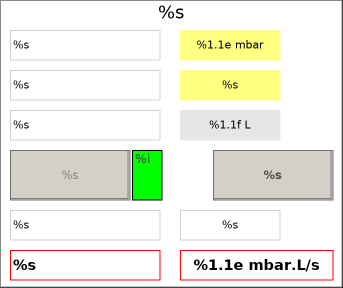
VISUALIZATION SA_TEST_RP  // 343x288
VAR_IN_OUT
	m_Input_Operation:		BLOCK_OPERATION;
	m_Input_Pression:		REAL;		(*PRM pression initiale*)
	m_Input_Duree:			TIME;		(*PRM temps du test*)
	m_Input_Volume:			REAL;		(*CONF volume*)
	m_Input_Co_Stop:		BOOL;		(*Co stop*)
	m_Input_Timer:			TIME;		(*Tps écoulé*)
	m_Input_Result:			REAL;		(*Résultat*)
END_VAR
    Rectangle (0,0 343x288), "%s", text list: 'TextList_Test_RP', text index: 0
    Textfield (10,30 150x30), "%s", text list: 'TextList_Test_RP', text index: 1
    Textfield (10,70 150x30), "%s", text list: 'TextList_Test_RP', text index: 2
    Textfield (10,110 150x30), "%s", text list: 'TextList_Test_RP', text index: 3
    Textfield (10,210 150x30), "%s", invisible if: m_Input_Operation.OK OR m_Input_Operation.AR, text list: 'TextList_Test_RP', text index: 4
    Textfield (10,250 150x30), "%s", invisible if: m_Input_Operation.EC, text list: 'TextList_Test_RP', text index: 5
    Textfield (180,30 100x30), "%1.1e mbar", text variable: m_Input_Pression, input disabled if: (NOT PRG_USER.ACTU_USER.FONCTION_SA AND NOT MACHINE.STATE_Prod) OR MACHINE.STATE_Prod
        OnMouseClick: write the text variable via InputWithLimits, min 0, max 1000
    Textfield (180,70 100x30), "%s", text variable: m_Input_Duree, input disabled if: (NOT PRG_USER.ACTU_USER.FONCTION_SA AND NOT MACHINE.STATE_Prod) OR MACHINE.STATE_Prod
        OnMouseClick: write the text variable via InputWithLimits
    Textfield (180,110 100x30), "%1.1f L", text variable: m_Input_Volume
    Frame (10,150 152x50)
        shows VISU_FCTS_SA(m_Input_ID_XML := 5, m_Input_UserRight := PRG_USER.ACTU_USER.FONCTION_SA AND NOT MACHINE.STATE_PROD, m_Input_Operation := m_Input_Operation)
    Button (213,150 120x50), "%s", input disabled if: NOT (PRG_User.ACTU_USER.FONCTION_SA AND NOT MACHINE.STATE_PROD), text list: 'TextList_Test_RP', text index: 6
        toggle m_Input_Co_Stop
    Textfield (180,210 100x30), "%s", text variable: m_Input_Timer, invisible if: m_Input_Operation.OK OR m_Input_Operation.AR
    Textfield (180,250 153x30), "%1.1e mbar.L/s", text variable: m_Input_Result, invisible if: m_Input_Operation.EC
END_VISUALIZATION

// ---- Visualizations/Semi Auto/Elements/SA_VERIN.TcVIS
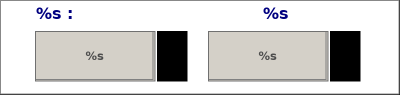
VISUALIZATION SA_VERIN  // 400x95
VAR_IN_OUT
	m_Input_VERIN : BLOCK_ACTUATOR;
END_VAR
    RoundedRectangle (0,0 400x95), text variable: m_Input_VERIN.MNEMO
    RoundedRectangle (157,31 30x50), colour toggle: m_Input_VERIN.STATE_ON
    Button (35,31 120x50), "%s", input disabled if: NOT m_Input_VERIN.Autor_On_IHM OR NOT m_Input_VERIN.MANUAL OR NOT (PRG_User.ACTU_USER.FONCTION_SA AND NOT MACHINE.STATE_PROD), text list: 'TextList_Orders', text index: 3
        tap m_Input_VERIN.M_ON
    RoundedRectangle (330,31 30x50), colour toggle: m_Input_VERIN.STATE_Off
    Button (208,31 120x50), "%s", input disabled if: NOT m_Input_VERIN.Autor_Off_IHM OR NOT m_Input_VERIN.MANUAL OR NOT (PRG_User.ACTU_USER.FONCTION_SA AND NOT MACHINE.STATE_PROD), text list: 'TextList_Orders', text index: 2
        tap m_Input_VERIN.M_OFF
    Rectangle (33,3 247x21), "%s :", text list: 'TextList_Actuator_Type', text index: 0
    Rectangle (260,3 119x21), "%s", text variable: m_Input_VERIN.MNEMO
END_VISUALIZATION

// ---- Visualizations/Semi Auto/VISU_SA.TcVIS
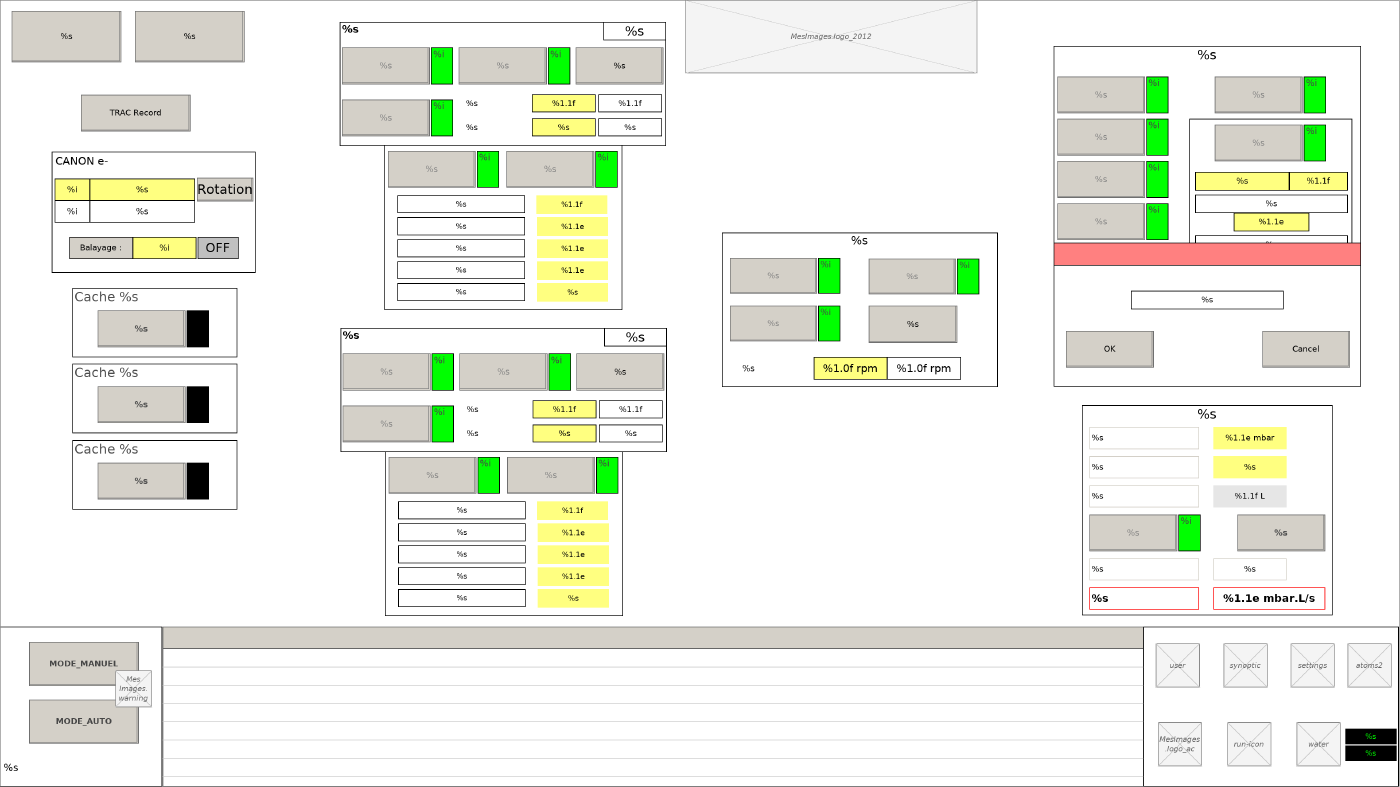
VISUALIZATION VISU_SA  // 1920x1080, background image fond_blanc_1280_1024
    Frame (223,860 1061x221)
        shows VISU_EV_EXTRAIT()
    Frame (1568,860 352x162)
        shows VISU_BANDEAU(m_Input_MACHINE := Global_Variables.MACHINE)
    Frame (0,860 221x162)
        shows VISU_MODE_MARCHE(m_Input_MACHINE := .MACHINE)
    Frame (71,208 284x138)
        shows SA_EVAP(m_Input_Crucible := PRG_EVAP.CRUCIBLE1, m_Input_Sweep := PRG_EVAP.SWEEP1)
    Frame (99,395 226x95)
        shows SA_CACHE_ACTUATOR(m_Input_CACHE := PRG_EVAP.CC11, m_Input_PRM_Forcage := PRG_EVAP.PRM_Forcage_Cache_Source1)
    Frame (466,30 447x170)
        shows SA_LIGNE_GAZ_MKS_RAMPE(m_Input_Ligne := PRG_GAZ.LIGNE_GAZ[1], m_Input_Machine := MACHINE, m_Input_DG := .PRG_GAZ.DG[1], m_Input_UserRight := PRG_USER.ACTU_USER.FONCTION_SA, m_Input_NumTextList := 11)
    Frame (99,499 226x95)
        shows SA_CACHE_ACTUATOR(m_Input_CACHE := PRG_EVAP.CC12, m_Input_PRM_Forcage := PRG_EVAP.PRM_Forcage_Cache_Source2)
    Frame (990,319 378x225)
        shows SA_ROT(m_Input_ROT := PRG_MOUVEMENT_PS.ROTATION_PS, m_Input_PRG := PRG_MOUVEMENT_PS)
    Frame (99,604 226x95)
        shows SA_CACHE_ACTUATOR(m_Input_CACHE := PRG_EVAP.CC13, m_Input_PRM_Forcage := PRG_EVAP.PRM_Forcage_Cache_Source3)
    Button (16,15 150x70), "%s", text list: 'TextList_Navigation', text index: 0
        OnMouseClick: change screen: SYN_POMPAGE
    Button (185,15 150x70), "%s", text list: 'TextList_Navigation', text index: 1
        OnMouseClick: change screen: SYN_PROC
    Frame (527,199 326x226)
        shows SA_REGUL_GAZ(m_Input_REGULATION := PRG_GAZ.REGULATION_GAZ_L1, m_Input_MACHINE := .MACHINE)
    Frame (528,619 326x226)
        shows SA_REGUL_GAZ(m_Input_REGULATION := PRG_GAZ.REGULATION_GAZ_L2, m_Input_MACHINE := .MACHINE)
    Frame (1484,556 344x289)
        shows SA_TEST_RP(m_Input_Operation := PRG_POMPAGE.POMPAGE.OP_Test_RP, m_Input_Pression := PRG_POMPAGE.POMPAGE.PRM_Pr_test, m_Input_Duree := PRG_POMPAGE.POMPAGE.PRM_Tim_test, m_Input_Volume := PRG_POMPAGE.POMPAGE.CONF_Volume_Enceinte, m_Input_Co_Stop := PRG_POMPAGE.POMPAGE.CO_Stop_Test_RP, m_Input_Timer := PRG_POMPAGE.POMPAGE.TIMER_attente_test.ET, m_Input_Result := PRG_POMPAGE.POMPAGE.VAR_Indicateur_Test)
    Frame (1445,63 422x467)
        shows SA_POMP_1E_PCR_PPM_ASS_M11(m_Input_PRG := PRG_POMPAGE, m_Input_Jauge := PRG_POMPAGE.M11, m_Input_Vanne := PRG_POMPAGE.POMPAGE.VS11, m_Input_Machine := MACHINE)
    Button (111,130 150x50), "TRAC Record", colour toggle: MAIN.Enr_TRAC
        toggle MAIN.Enr_TRAC
    Frame (467,450 447x170)
        shows SA_LIGNE_GAZ_MKS_RAMPE(m_Input_Ligne := PRG_GAZ.LIGNE_GAZ[2], m_Input_Machine := MACHINE, m_Input_DG := .PRG_GAZ.DG[2], m_Input_UserRight := PRG_USER.ACTU_USER.FONCTION_SA, m_Input_NumTextList := 12)
    Image (940,0 400x100), image: MesImages.logo_2012
END_VISUALIZATION

// ---- Visualizations/Symbole/CACHE/SYM_CACHE.TcVIS
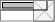
VISUALIZATION SYM_CACHE  // 55x22
VAR_IN_OUT
	m_Input_CACHE : BLOCK_ACTUATOR;
END_VAR
    Rectangle (2,2 43x6), colour toggle: (m_Input_CACHE.STATE_OFF) <> 0, invisible if: (m_Input_CACHE.STATE_ON) <> 0
    Rectangle (0,0 47x10), invisible if: NOT m_Input_CACHE.AUTOR_On_IHM OR NOT PRG_USER.ACTU_USER.MAINTENANCE, input disabled if: NOT m_Input_CACHE.AUTOR_On_IHM OR NOT PRG_User.ACTU_USER.MAINTENANCE
        tap m_Input_CACHE.M_ON
    Image (33,0 22x22), invisible if: NOT m_Input_CACHE.STATE_NOK, image: MesImages.warning
    Rectangle (0,0 47x10), invisible if: NOT m_Input_CACHE.AUTOR_Off_IHM OR NOT PRG_USER.ACTU_USER.MAINTENANCE, input disabled if: NOT m_Input_CACHE.AUTOR_Off_IHM OR NOT PRG_User.ACTU_USER.MAINTENANCE
        tap m_Input_CACHE.M_Off
END_VISUALIZATION

// ---- Visualizations/Symbole/CACHE/SYM_CACHE_ACTUATOR2.TcVIS
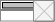
VISUALIZATION SYM_CACHE_ACTUATOR2  // 55x22
VAR_IN_OUT
	m_Input_CACHE : BLOCK_ACTUATOR2;
END_VAR
    Rectangle (2,2 43x6), colour toggle: (m_Input_CACHE.STATE_OFF) <> 0, invisible if: (m_Input_CACHE.STATE_ON) <> 0
    Rectangle (0,0 47x10), invisible if: NOT m_Input_CACHE.AUTOR_On_IHM AND NOT m_Input_CACHE.AUTOR_Off_IHM OR NOT PRG_USER.ACTU_USER.MAINTENANCE, input disabled if: NOT m_Input_CACHE.AUTOR_On_IHM AND NOT m_Input_CACHE.AUTOR_Off_IHM OR NOT PRG_User.ACTU_USER.MAINTENANCE
        tap m_Input_CACHE.M_ON
    Image (33,0 22x22), invisible if: NOT m_Input_CACHE.STATE_NOK, image: MesImages.warning
END_VISUALIZATION

// ---- Visualizations/Symbole/Chauffage/VISU_CHAUFF.TcVIS
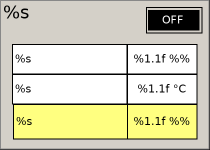
VISUALIZATION VISU_CHAUFF  // 210x150
VAR_IN_OUT
	m_Input_ELMT_CHAUFF:	BLOCK_ELMT_CHAUFF;
END_VAR
    Rectangle (0,0 210x150), "%s", text list: 'TextList_Chauffage', text index: 0
    RoundedRectangle (12,44 115x30), "%s", text list: 'TextList_Chauffage', text index: 1
    RoundedRectangle (127,44 70x30), "%1.1f %%", text variable: m_Input_ELMT_CHAUFF.OUT_QCH.Value
    RoundedRectangle (149,10 50x20), "ON", invisible if: NOT m_Input_ELMT_CHAUFF.OUT_MCH
    RoundedRectangle (148,10 50x20), "OFF", invisible if: m_Input_ELMT_CHAUFF.OUT_MCH
    RoundedRectangle (13,104 116x35), "%s", invisible if: NOT m_Input_ELMT_CHAUFF.PRM_Ctrl, input disabled if: NOT m_Input_ELMT_CHAUFF.MANUAL OR NOT PRG_USER.ACTU_USER.MAINTENANCE, text list: 'TextList_Chauffage', text index: 3
        OnMouseClick: toggle m_Input_ELMT_CHAUFF.PRM_Ctrl
    RoundedRectangle (127,104 70x35), "%1.1f °C", text variable: m_Input_ELMT_CHAUFF.PRM_Temperature, invisible if: NOT m_Input_ELMT_CHAUFF.PRM_Ctrl, input disabled if: NOT m_Input_ELMT_CHAUFF.MANUAL OR NOT PRG_USER.ACTU_USER.MAINTENANCE
        OnMouseClick: write the text variable via VisuDialogs.Numpad, min m_Input_ELMT_CHAUFF.CONF_TMIN, max m_Input_ELMT_CHAUFF.CONF_TMAX
    RoundedRectangle (127,74 70x30), "%1.1f °C", text variable: m_Input_ELMT_CHAUFF.IN_Temperature
    RoundedRectangle (12,74 115x30), "%s", text list: 'TextList_Chauffage', text index: 2
    RoundedRectangle (13,104 115x35), "%s", invisible if: m_Input_ELMT_CHAUFF.PRM_Ctrl, input disabled if: NOT m_Input_ELMT_CHAUFF.MANUAL OR NOT PRG_USER.ACTU_USER.MAINTENANCE, text list: 'TextList_Chauffage', text index: 4
        OnMouseClick: toggle m_Input_ELMT_CHAUFF.PRM_Ctrl
    RoundedRectangle (127,104 70x35), "%1.1f %%", text variable: m_Input_ELMT_CHAUFF.PRM_Power, invisible if: m_Input_ELMT_CHAUFF.PRM_Ctrl, input disabled if: NOT m_Input_ELMT_CHAUFF.MANUAL OR NOT PRG_USER.ACTU_USER.MAINTENANCE
        OnMouseClick: write the text variable via VisuDialogs.Numpad, min 0, max m_Input_ELMT_CHAUFF.CONF_PMAX
    Rectangle (146,7 56x26), invisible if: (NOT m_Input_ELMT_CHAUFF.AUTOR_Off_IHM AND NOT m_Input_ELMT_CHAUFF.AUTOR_On_IHM) OR NOT PRG_USER.ACTU_USER.MAINTENANCE, input disabled if: (NOT m_Input_ELMT_CHAUFF.AUTOR_Off_IHM AND NOT m_Input_ELMT_CHAUFF.AUTOR_On_IHM) OR NOT PRG_USER.ACTU_USER.MAINTENANCE
        tap m_Input_ELMT_CHAUFF.M_On
END_VISUALIZATION

// ---- Visualizations/Symbole/Chauffage/VISU_CONFIG_CHAUFF.TcVIS
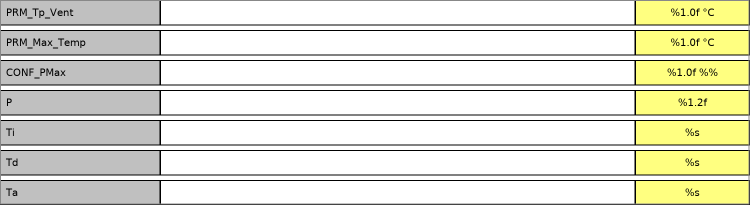
VISUALIZATION VISU_CONFIG_CHAUFF  // 750x205
(*visualistion pour secondaire dans chambre et primaire dans sas ==> paramètres pour chambre*)
VAR_IN_OUT
	m_Input_PRG_CHAUFFAGE : BLOCK_PRG_CHAUFFAGE;
END_VAR
    Rectangle (160,0 475x25), text list: 'TextList_Config_Chauffage', text index: 1
    Rectangle (635,0 115x25), "%1.0f °C", text variable: m_Input_PRG_CHAUFFAGE.PRM_Tp_Vent, input disabled if: NOT Global_Variables.PRG_USER.ACTU_USER.CONF_MACHINE
        OnMouseClick: write the text variable via VisuDialogs.Numpad, min m_Input_PRG_CHAUFFAGE.CONF_Min_Temp, max 55
    Rectangle (0,0 160x25), "PRM_Tp_Vent"
    Rectangle (160,30 475x25), text list: 'TextList_Config_Chauffage', text index: 2
    Rectangle (635,30 115x25), "%1.0f °C", text variable: m_Input_PRG_CHAUFFAGE.PRM_Max_Temp, input disabled if: NOT Global_Variables.PRG_USER.ACTU_USER.CONF_MACHINE
        OnMouseClick: write the text variable via VisuDialogs.Numpad, min m_Input_PRG_CHAUFFAGE.CONF_Min_Temp, max m_Input_PRG_CHAUFFAGE.CONF_Max_Temp
    Rectangle (0,30 160x25), "PRM_Max_Temp"
    Rectangle (160,60 475x25), text list: 'TextList_Config_Chauffage', text index: 3
    Rectangle (160,90 475x25), text list: 'TextList_Config_Chauffage', text index: 4
    Rectangle (635,60 115x25), "%1.0f %%", text variable: m_Input_PRG_CHAUFFAGE.CHAUFFAGE.CH.CONF_PMAX, input disabled if: NOT Global_Variables.PRG_USER.ACTU_USER.CONF_MACHINE
        OnMouseClick: write the text variable via VisuDialogs.Numpad, min 0, max m_Input_PRG_CHAUFFAGE.CONF_Pmax_max
    Rectangle (0,60 160x25), "CONF_PMax"
    Rectangle (635,90 115x25), "%1.2f", text variable: m_Input_PRG_CHAUFFAGE.CHAUFFAGE.CH.PRM_PID.KpHeat, input disabled if: NOT Global_Variables.PRG_USER.ACTU_USER.CONF_MACHINE
        OnMouseClick: write the text variable via VisuDialogs.Numpad, min 0
    Rectangle (0,90 160x25), "P"
    Rectangle (160,120 475x25), text list: 'TextList_Config_Chauffage', text index: 5
    Rectangle (635,120 115x25), "%s", text variable: m_Input_PRG_CHAUFFAGE.CHAUFFAGE.CH.PRM_PID.TnHeat, input disabled if: NOT Global_Variables.PRG_USER.ACTU_USER.CONF_MACHINE
        OnMouseClick: write the text variable via VisuDialogs.Keypad
    Rectangle (0,120 160x25), "Ti"
    Rectangle (0,150 160x25), "Td"
    Rectangle (160,150 475x25), text list: 'TextList_Config_Chauffage', text index: 6
    Rectangle (635,150 115x25), "%s", text variable: m_Input_PRG_CHAUFFAGE.CHAUFFAGE.CH.PRM_PID.TvHeat, input disabled if: NOT Global_Variables.PRG_USER.ACTU_USER.CONF_MACHINE
        OnMouseClick: write the text variable via VisuDialogs.Keypad
    Rectangle (0,180 160x25), "Ta"
    Rectangle (160,180 475x25), text list: 'TextList_Chauffage', text index: 6
    Rectangle (635,180 115x25), "%s", text variable: m_Input_PRG_CHAUFFAGE.CHAUFFAGE.CH.PRM_PID.TdHeat, input disabled if: NOT Global_Variables.PRG_USER.ACTU_USER.CONF_MACHINE
        OnMouseClick: write the text variable via VisuDialogs.Keypad
END_VISUALIZATION

// ---- Visualizations/Symbole/Chauffage/VISU_LAMPE.TcVIS
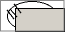
VISUALIZATION VISU_LAMPE  // 65x32
VAR_IN_OUT
	m_Input_ELMT_CHAUFF:	BLOCK_ELMT_CHAUFF;
END_VAR
    Ellipse (7,1 50x30), angle 331, colour toggle: m_Input_ELMT_CHAUFF.OUT_MCH
    Rectangle (15,8 50x24), angle 330
    Group (7,4 14x15), invisible if: NOT m_Input_ELMT_CHAUFF.OUT_MCH
        Line (7,15) (0,6)
        Line (10,13) (3,5)
        Line (14,9) (7,0)
END_VISUALIZATION

// ---- Visualizations/Symbole/DIVERS/CHRONO.TcVIS
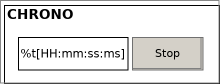
VISUALIZATION CHRONO  // 220x84
VAR_IN_OUT
	m_input_CHRONO : TON;
END_VAR
    Rectangle (4,5 216x79), "CHRONO"
    RoundedRectangle (18,37 110x33), "%t[HH:mm:ss:ms]", text variable: m_input_CHRONO.ET
        OnMouseDown: write the text variable via VisuDialogs.Numpad, min 7, max 10
    Button (132,37 71x33), "Start", invisible if: m_input_CHRONO.IN
        OnMouseClick: execute { m_input_CHRONO.IN := TRUE; }
    Button (132,37 71x33), "Stop", invisible if: NOT m_input_CHRONO.IN
        OnMouseClick: execute { m_input_CHRONO.IN := FALSE; }
END_VISUALIZATION

// ---- Visualizations/Symbole/Effluvage/VISU_CONFIG_EFF.TcVIS
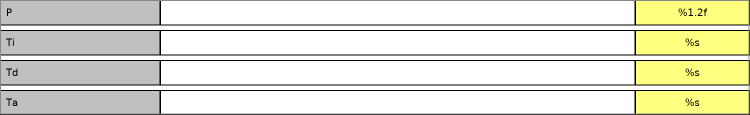
VISUALIZATION VISU_CONFIG_EFF  // 750x115
VAR_IN_OUT
	m_Input_PRG_EFFLUVAGE : BLOCK_PRG_EFFLUVAGE;
END_VAR
    Rectangle (160,0 475x25), text list: 'TextList_Config_EFFLUVAGE', text index: 4
    Rectangle (635,0 115x25), "%1.2f", text variable: m_Input_PRG_EFFLUVAGE.Effluvage.ALEFF.CONF_Kp, input disabled if: NOT Global_Variables.PRG_USER.ACTU_USER.CONF_MACHINE
        OnMouseClick: write the text variable via InputWithLimits, min 0
    Rectangle (0,0 160x25), "P"
    Rectangle (160,30 475x25), text list: 'TextList_Config_EFFLUVAGE', text index: 5
    Rectangle (635,30 115x25), "%s", text variable: m_Input_PRG_EFFLUVAGE.Effluvage.ALEFF.CONF_Tn, input disabled if: NOT Global_Variables.PRG_USER.ACTU_USER.CONF_MACHINE
        OnMouseClick: write the text variable via InputWithLimits
    Rectangle (0,30 160x25), "Ti"
    Rectangle (0,60 160x25), "Td"
    Rectangle (160,60 475x25), text list: 'TextList_Config_EFFLUVAGE', text index: 6
    Rectangle (635,60 115x25), "%s", text variable: m_Input_PRG_EFFLUVAGE.Effluvage.ALEFF.CONF_Tv, input disabled if: NOT Global_Variables.PRG_USER.ACTU_USER.CONF_MACHINE
        OnMouseClick: write the text variable via InputWithLimits
    Rectangle (0,90 160x25), "Ta"
    Rectangle (160,90 475x25), text list: 'TextList_Config_EFFLUVAGE', text index: 7
    Rectangle (635,90 115x25), "%s", text variable: m_Input_PRG_EFFLUVAGE.Effluvage.ALEFF.CONF_Td, input disabled if: NOT Global_Variables.PRG_USER.ACTU_USER.CONF_MACHINE
        OnMouseClick: write the text variable via InputWithLimits
END_VISUALIZATION

// ---- Visualizations/Symbole/Effluvage/VISU_EFFLUVAGE.TcVIS
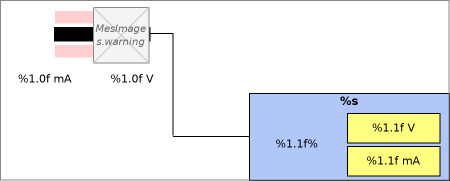
VISUALIZATION VISU_EFFLUVAGE  // 450x181
VAR_IN_OUT
	M_input_effluvage:	BLOCK_PRG_EFFLUVAGE;
END_VAR
    Line (140,33) (173,33)
    Line (173,136) (324,136)
    RoundedRectangle (55,11 93x12), invisible if: NOT M_input_effluvage.Effluvage.ALEFF.STATE_plasma
    Rectangle (2,64 86x30), "%1.0f mA", text variable: M_input_effluvage.Effluvage.ALEFF.STATE_current, invisible if: M_input_effluvage.Effluvage.ALEFF.STATE_OFF
    Rectangle (89,64 86x30), "%1.0f V", text variable: M_input_effluvage.Effluvage.ALEFF.STATE_tension, invisible if: M_input_effluvage.Effluvage.ALEFF.STATE_OFF
    RoundedRectangle (249,93 201x88), "%s", text list: 'TextList_Effluvage', text index: 1
    Textfield (257,132 80x24), "%1.1f%", text variable: M_input_effluvage.Effluvage.ALEFF.STATE_Setpoint_Power
    Rectangle (347,113 93x30), "%1.1f V", text variable: M_input_effluvage.Effluvage.PRM_Tension_attendue, invisible if: NOT M_input_effluvage.Effluvage.MANUAL, input disabled if: NOT PRG_USER.ACTU_USER.MAINTENANCE OR NOT PRG_EFFLUVAGE.Effluvage.Manual
        OnMouseClick: write the text variable via InputWithLimits, min 0, max M_input_effluvage.Effluvage.ALEFF.IN_CURRENT.CONF_Max
    RoundedRectangle (55,45 93x12), invisible if: NOT M_input_effluvage.Effluvage.ALEFF.STATE_plasma
    RoundedRectangle (54,27 96x14), colour toggle: PRG_EFFLUVAGE.Effluvage.ALEFF.STATE_ON, input disabled if: NOT PRG_USER.ACTU_USER.MAINTENANCE OR NOT PRG_EFFLUVAGE.Effluvage.Manual
        OnMouseClick: toggle M_input_effluvage.Effluvage.ALEFF.M_ON
    Image (93,7 56x56), invisible if: NOT M_input_effluvage.Effluvage.ALEFF.STATE_NOK, image: MesImages.warning
    Line (173,135) (173,33)
    Rectangle (347,146 93x30), "%1.1f mA", text variable: M_input_effluvage.Effluvage.PRM_consigne, invisible if: NOT M_input_effluvage.Effluvage.MANUAL, input disabled if: NOT PRG_USER.ACTU_USER.MAINTENANCE OR NOT PRG_EFFLUVAGE.Effluvage.Manual
        OnMouseClick: write the text variable via InputWithLimits, min 0, max M_input_effluvage.Effluvage.ALEFF.IN_CURRENT.CONF_Max
END_VISUALIZATION

// ---- Visualizations/Symbole/EVAP/VISU_ALIM_HT.TcVIS
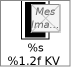
VISUALIZATION VISU_ALIM_HT  // 71x67
VAR_IN_OUT
	m_Input_HT:				BLOCK_HT_CANON_ST10;
END_VAR
VAR_IN_OUT
	m_Input_NO_HV_RET:		BOOL;
END_VAR
    Rectangle (25,2 20x35), colour toggle: m_Input_HT.STATE_HV_ON, invisible if: NOT m_Input_HT.STATE_HV_ON AND NOT m_Input_HT.STATE_HV
    Rectangle (25,2 20x35), invisible if: m_Input_HT.STATE_HV_ON OR m_Input_HT.STATE_HV
    Polygon (41,73)
    Rectangle (21,0 28x39), invisible if: NOT m_Input_HT.HV.AUTOR_On_IHM AND NOT m_Input_HT.HV.AUTOR_Off_IHM, input disabled if: (NOT m_Input_HT.HV.AUTOR_ON_IHM AND NOT m_Input_HT.HV.AUTOR_OFF_IHM) OR NOT PRG_User.ACTU_USER.MAINTENANCE
        tap m_Input_HT.HV.M_On
    Rectangle (0,41 71x14), "%s", text variable: m_Input_HT.MNEMO
    Rectangle (0,55 71x12), "%1.2f KV", text variable: m_Input_HT.STATE_V_HV, invisible if: (m_Input_NO_HV_RET) <> 0
    Image (31,4 29x28), invisible if: NOT m_Input_HT.STATE_NOK, image: MesImages.warning
END_VISUALIZATION

// ---- Visualizations/Symbole/EVAP/VISU_ALIM_HT_S10.TcVIS
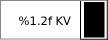
VISUALIZATION VISU_ALIM_HT_S10  // 108x40
VAR_IN_OUT
	m_Input_HT:				BLOCK_CANON_ST10;
END_VAR
VAR_IN_OUT
END_VAR
    Rectangle (84,2 20x35), colour toggle: m_Input_HT.STATE_HV_ON, invisible if: NOT m_Input_HT.STATE_HV_ON AND NOT m_Input_HT.STATE_HV
    Rectangle (84,2 20x35), invisible if: m_Input_HT.STATE_HV_ON OR m_Input_HT.STATE_HV
    Polygon (41,73)
    Rectangle (80,0 28x40), invisible if: NOT m_Input_HT.HV.AUTOR_On_IHM AND NOT m_Input_HT.HV.AUTOR_Off_IHM, input disabled if: (NOT m_Input_HT.HV.AUTOR_ON_IHM AND NOT m_Input_HT.HV.AUTOR_OFF_IHM) OR NOT PRG_User.ACTU_USER.MAINTENANCE
        tap m_Input_HT.HV.M_On
    Rectangle (11,15 71x12), "%1.2f KV", text variable: m_Input_HT.STATE_V_HV
END_VISUALIZATION

// ---- Visualizations/Symbole/EVAP/VISU_BAL_MANU.TcVIS
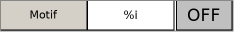
VISUALIZATION VISU_BAL_MANU  // 234x32
VAR_IN_OUT
	m_Input_BAL: BLOCK_TELEMARK_DIGITAL_SWEEP;
END_VAR
    Rectangle (87,0 87x30), "%i", text variable: m_Input_BAL.PRM_NbBal, input disabled if: NOT (Global_Variables.PRG_USER.ACTU_USER.FONCTION_SA AND NOT MACHINE.STATE_PROD)
        OnMouseClick: write the text variable via VisuDialogs.Numpad, min 1, max 8
    RoundedRectangle (176,0 56x30), "ON", invisible if: NOT m_Input_BAL.STATE_ON
    RoundedRectangle (176,0 56x30), "OFF", invisible if: NOT m_Input_BAL.STATE_OFF
    Rectangle (0,0 87x30), "Motif"
END_VISUALIZATION

// ---- Visualizations/Symbole/EVAP/VISU_CANON.TcVIS
